FUNCTION fBoolToText  : STRING
VAR_INPUT
    bValue : BOOL;
END_VAR

IF bValue THEN
    fBoolToText := 'TRUE';
ELSE
    fBoolToText := 'FALSE';
END_IF

END_FUNCTION

(* stored: Version 1.1.0.1, ProductVersion 3.1.4024.15
   POU fBoolToText: Id {b4e1153d-e370-4b2b-8839-e8f8c6c28b67}, SpecialFunc None *)
